// Mitsubishi GX Works2 project: timer01   PLC: Q02/Q02H

PROGRAM MAIN
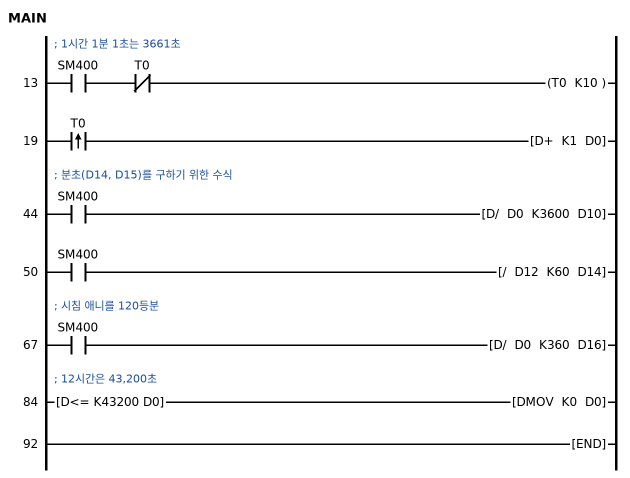
; 1시간 1분 1초는 3661초
13    LD      SM400
      ANI     T0
      OUT     T0 K10
19    LDP     T0
      D+      K1 D0
; 분초(D14, D15)를 구하기 위한 수식
44    LD      SM400
      D/      D0 K3600 D10
50    LD      SM400
      /       D12 K60 D14
; 시침 애니를 120등분
67    LD      SM400
      D/      D0 K360 D16
; 12시간은 43,200초
84    LDD<=   K43200 D0
      DMOV    K0 D0
92    END
END_PROGRAM
